FUNCTION_BLOCK 
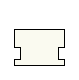
  EVENT_INPUT
    ;
  END_EVENT
  EVENT_OUTPUT
    ;
  END_EVENT
  VAR_INPUT
     : ;
     : ;
  END_VAR
  VAR_OUTPUT
     : ;
     : ;
     : ;
     : ;
  END_VAR
  ALGORITHM ALG IN ST:

  END_ALGORITHM
END_FUNCTION_BLOCK
(* other elements stored in the file *)
(* ECState name=START Initial=true *)
(* ECState name=BODY *)
(* ECAction Algorithm=ALG *)
(* ECTransition Source=START Destination=BODY *)
(* ECEventCondition Event=EP1 *)
(* ECTransition Source=BODY Destination=EP2_STATE *)
(* ECCondition  (LS >= LS2) *)
(* ECState Name=EP2_STATE *)
(* ECAction Output=EP2 *)
